ABB RobotStudio station: Proyecto Final.rsstn

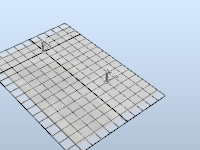
Station Station (saved by RobotStudio 20.4.9280.0)
Controller IRB4600_40_255_Inicial, task T_ROB1: task frame (RAPID world) sits at (8000, 2000, 0) mm in the station
Controller IRB4600_40_255_Inicial
  mechanical unit ROB_1: IRB4600_40_255_C_01, 6 joints, base frame (0, 0, 0) mm
Controller IRB4600_40_255_Final
  mechanical unit ROB_1: IRB4600_40_255_C_01_2, 6 joints, base frame (0, 0, 0) mm
Controller IRB2600_12_165
  mechanical unit ROB_1: IRB2600_12_165_C_01, 6 joints, base frame (0, 0, 0) mm
Layout (positions relative to the parent item):
  - IRB4600_40_255_C_01 [mechanism, from Robots\IRB4600_40_255_C_G_01.rslib] at (8000, 2000, 0) mm; joint values [0, 0, 0, 0, 0.5236, 0] (rad or m)
  - IRB4600_40_255_C_01_2 [mechanism, from Robots\IRB4600_40_255_C_G_01.rslib] at (0, 0, 0) mm; joint values [0, 0, 0, 0, 0.5236, 0] (rad or m)
  - IRB2600_12_165_C_01 [mechanism, from Robots\IRB2600_12_165_C_01.rslib] at (0, 0, 0) mm; joint values [0, 0, 0, 0, 0.5236, 0] (rad or m)
  - Floor [part]
